{attribute 'qualified_only'}
VAR_GLOBAL
	pMainJibCylinder : ST_pValveControlledCylinder;
	pMainKnuckleCylinder : ST_pValveControlledCylinder;
END_VAR

(* stored: Version 1.1.0.1, ProductVersion 3.1.4024.9
   GVL Param: Id {8cc71902-54f3-4068-b684-2ff92871ee93} *)
